FUNCTION_BLOCK HWMsg (* Basic FB with empty ECC *)
  (* Standard: 61499-2 *)
  (* Version 1.0, 2021-03-18, AK120569 *)
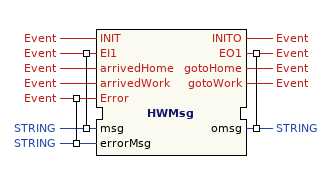
  EVENT_INPUT
    INIT;
    EI1 WITH msg;
    arrivedHome;
    arrivedWork;
    Error WITH errorMsg;
  END_EVENT
  EVENT_OUTPUT
    INITO;
    EO1 WITH omsg;
    gotoHome;
    gotoWork;
  END_EVENT
  VAR_INPUT
    msg : STRING;
    errorMsg : STRING;
  END_VAR
  VAR_OUTPUT
    omsg : STRING;
  END_VAR
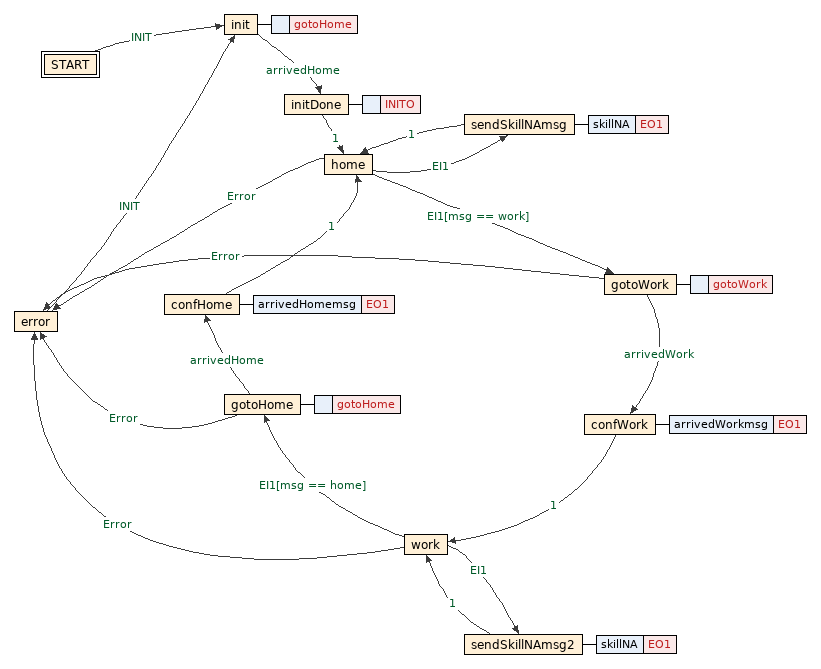
  EC_STATES
    START; (* Initial State *)
    home;
    init : -> gotoHome;
    work;
    gotoWork : -> gotoWork;
    gotoHome : -> gotoHome;
    error;
    sendSkillNAmsg : skillNA -> EO1;
    sendSkillNAmsg2 : skillNA -> EO1;
    confWork : arrivedWorkmsg -> EO1;
    confHome : arrivedHomemsg -> EO1;
    initDone : -> INITO;
  END_STATES
  EC_TRANSITIONS
    START TO init := INIT;
    home TO gotoWork := EI1[msg ==  work];
    work TO gotoHome := EI1[msg  == home];
    error TO init := INIT;
    gotoHome TO error := Error;
    home TO error := Error;
    work TO error := Error;
    gotoWork TO error := Error;
    home TO sendSkillNAmsg := EI1;
    sendSkillNAmsg TO home := 1;
    work TO sendSkillNAmsg2 := EI1;
    sendSkillNAmsg2 TO work := 1;
    gotoWork TO confWork := arrivedWork;
    confWork TO work := 1;
    gotoHome TO confHome := arrivedHome;
    confHome TO home := 1;
    init TO initDone := arrivedHome;
    initDone TO home := 1;
  END_TRANSITIONS
  ALGORITHM skillNA IN ST:
omsg := "NA";
  END_ALGORITHM
  ALGORITHM arrivedWorkmsg IN ST:
omsg := "work";
  END_ALGORITHM
  ALGORITHM arrivedHomemsg IN ST:
omsg := "home";
  END_ALGORITHM
END_FUNCTION_BLOCK
